INTERFACE ITF_SPM_HMI_Init EXTENDS B_Baza.ITF_PodzespolBazowy, ITF_SPM_HMI_Lacznik

END_INTERFACE

(* stored: Version 1.1.0.1
   Itf ITF_SPM_HMI_Init: Id {fc6e9688-124c-4b91-a404-07682a7daf92} *)
